TYPE MachineSectionHMIInterface :
STRUCT
	ActiveMachineSection : MachineSection;
	SelectedActor : INT;
	PageSwitch	:	HMIWindowSwitch;
	Movements : HMIMovementInterface;
	Forks : HMIMovementForkInterface;
	Runcontrols : HMIRuncontrolInterface;
	RFID : HMIRFIDInterface;
	Workpiece : HMIWorkpieceInterface;
END_STRUCT
END_TYPE

(* stored: Version 1.1.0.1
   DUT MachineSectionHMIInterface: Id {0ed9cdeb-5e9f-436a-94ad-dc91dcd1c0be} *)
